INTERFACE ITFModule

METHOD M_Abort
END_METHOD

METHOD M_Hold
END_METHOD

METHOD M_Home
END_METHOD

METHOD M_Start
END_METHOD

METHOD M_Stop
END_METHOD

{attribute 'monitoring' := 'variable'}
PROPERTY PropBusy : BOOL
GET
END_GET
END_PROPERTY

{attribute 'monitoring' := 'variable'}
PROPERTY PropCurrentState : PACK_ML.State
GET
END_GET
END_PROPERTY

{attribute 'monitoring' := 'variable'}
PROPERTY PropErrDescription : STRING
GET
END_GET
END_PROPERTY

{attribute 'monitoring' := 'variable'}
PROPERTY PropError : BOOL
GET
END_GET
END_PROPERTY

END_INTERFACE

(* stored: Version 1.1.0.1
   Itf ITFModule: Id {83e2f220-b628-4cc1-8425-5ccb3ca1431d}
   Method M_Abort: Id {d4b36388-2c40-4a2a-840c-a7558cccf32c}
   Method M_Hold: Id {74dca715-0832-4e57-bd11-fa5482a40ca4}
   Method M_Home: Id {fa5ae12d-e278-43b8-b9fb-522a2f8363df}
   Method M_Start: Id {ede511b9-4a8a-4fd7-9a81-92329944db01}
   Method M_Stop: Id {b5172065-9e2b-4628-992b-67cbdd66121e}
   Property PropBusy: Id {826777bf-f2fe-40ca-a5f3-f2f24fef4c48}
   Get Get: Id {b22156fd-0bba-43bb-9a3c-a1c235b43373}
   Property PropCurrentState: Id {4900066d-af26-4295-98da-8b49be553787}
   Get Get: Id {eceb2763-c94a-4b06-ab47-cf1e57e608a6}
   Property PropErrDescription: Id {c91c07e4-f8e0-4585-a6d3-d7b49542a264}
   Get Get: Id {92d8f1b7-2d36-49bc-82dd-dd7e52bb62cc}
   Property PropError: Id {8b3b149d-5bc9-492d-bf03-7c656df23d5f}
   Get Get: Id {1d81e6fc-0e7b-4208-b519-b688ac452eb3} *)
